FUNCTION_BLOCK DisableGroupTask_TestSuite
VAR
	ThisTestSuite : TestSuite<TestSuiteParameter.MaxTestCount>('C:\ProgramData\Beckhoff\TwinCAT\3.1\Boot\DisableGroup_Tests.xml') := (TestSuiteName := 'DisableGroup Test Suite');
END_VAR

TaskAcceptsCommand_Test();
TaskRejectsDuplicateCommand_test();
TaskAcceptsValidCAGroup();
TaskRejectsExecuteWithNoCAGroup_Test();
TaskRejectsInvalidCAGroup();

METHOD TaskAcceptsCommand_Test
VAR
	stubCAGroup : CollisionGroup;
	testDisableGrp : DisableGroup := (MyCollisionGroup := stubCAGroup);
	Expected : BOOL := TRUE;
	Actual	 : BOOL;
END_VAR
IF ThisTestSuite.Test(__POUNAME()).ExecuteTest() THEN
	Actual := SUCCEEDED(testDisableGrp.Execute());
	testDisableGrp.Abort();
	ThisTestSuite.Test(__POUNAME()).AssertEqual(Expected, Actual);
END_IF
END_METHOD

METHOD TaskAcceptsValidCAGroup
VAR
	stubCAGroup : CollisionGroup;
	istuibCAGroup : I_CollisionGroup := stubCAGroup;
	testDisableGrp : DisableGroup := (MyCollisionGroup := stubCAGroup);
	Expected : BOOL := TRUE;
	Actual	 : BOOL;
END_VAR
IF ThisTestSuite.Test(__POUNAME()).ExecuteTest() THEN
	testDisableGrp.MyCollisionGroup := stubCAGroup;
	Actual := testDisableGrp.MyCollisionGroup = istuibCAGroup;
	ThisTestSuite.Test(__POUNAME()).AssertEqual(Expected, Actual);
END_IF
END_METHOD

METHOD TaskRejectsDuplicateCommand_test
VAR
	stubCAGroup : CollisionGroup;
	testDisableGrp : DisableGroup := (MyCollisionGroup := stubCAGroup);
	Expected : BOOL := TRUE;
	Actual	 : BOOL;
END_VAR
IF ThisTestSuite.Test(__POUNAME()).ExecuteTest() THEN
	testDisableGrp.Execute();
	Actual := FAILED(testDisableGrp.Execute());
	testDisableGrp.Abort();
	ThisTestSuite.Test(__POUNAME()).AssertEqual(Expected, Actual);
END_IF
END_METHOD

METHOD TaskRejectsExecuteWithNoCAGroup_Test
VAR
	testDisableGrp : DisableGroup ;
	Expected : BOOL := TRUE;
	Actual	 : BOOL;
END_VAR
IF ThisTestSuite.Test(__POUNAME()).ExecuteTest() THEN
	Actual := FAILED(testDisableGrp.Execute());
	testDisableGrp.Abort();
	ThisTestSuite.Test(__POUNAME()).AssertEqual(Expected, Actual);
END_IF
END_METHOD

METHOD TaskRejectsInvalidCAGroup
VAR
	stubCAGroup : CollisionGroup;
	iStubCAGroup : I_CollisionGroup := stubCAGroup;
	testDisableGrp : DisableGroup := (MyCollisionGroup := stubCAGroup);
	Expected : BOOL := TRUE;
	Actual	 : BOOL;
END_VAR
IF ThisTestSuite.Test(__POUNAME()).ExecuteTest() THEN
	testDisableGrp.MyCollisionGroup := 16#0;
	Actual := testDisableGrp.MyCollisionGroup = iStubCAGroup;
	ThisTestSuite.Test(__POUNAME()).AssertEqual(Expected, Actual);
END_IF
END_METHOD

END_FUNCTION_BLOCK

(* stored: Version 1.1.0.1
   POU DisableGroupTask_TestSuite: Id {408f9e89-352c-467f-9f88-651a03342266}, SpecialFunc None
   Method TaskAcceptsCommand_Test: Id {2f19c452-382f-4f73-9347-4d3d1fb24efb}
   Method TaskAcceptsValidCAGroup: Id {87defde3-5349-43fa-9862-fb8563ea554f}
   Method TaskRejectsDuplicateCommand_test: Id {e16752d3-6aa1-4e8c-94cf-e7f91998e657}
   Method TaskRejectsExecuteWithNoCAGroup_Test: Id {074498f0-77cd-499c-8ca0-4825d67d5d2b}
   Method TaskRejectsInvalidCAGroup: Id {b660fc48-6430-4c51-a2cb-f51c29cee9b7} *)
